(* IEC 61131-3 sources: Industrial-Automation-Portfolio/01_CONTROL_PLC/PLC-001_Automated_Conveyor_Control_System/02_IMPLEMENTATION/PLC/src, 1 file *)

(* ---- PLC001_Main.st ---- *)
(*
 PLC-001 — Automated Conveyor Control System
 Software-only portfolio implementation skeleton.

 Do not interpret this file as field-commissioned control code.
*)

TYPE E_MachineState :
(
    IDLE,
    RUNNING,
    TRANSFER,
    STOPPING,
    FAULT,
    E_STOP
);
END_TYPE

VAR
    State : E_MachineState := IDLE;
    StartCmd : BOOL;
    StopCmd : BOOL;
    EStopHealthy : BOOL;
    ProductDetected : BOOL;
    CriticalFault : BOOL;
    ResetCmd : BOOL;

    MotorRun : BOOL;
    FaultAlarm : BOOL;
END_VAR

(* Sequence logic to be completed and verified against test cases. *)
